FUNCTION_BLOCK DataConversionDecorator IMPLEMENTS ITF_Analogue
VAR
	wrappee : ITF_Analogue;
END_VAR

METHOD GetValue : INT
IF (THIS^.wrappee <> 0) THEN
  GetValue := THIS^.wrappee.GetValue() + 0.9;
END_IF
END_METHOD

END_FUNCTION_BLOCK

(* stored: Version 1.1.0.1, ProductVersion 3.1.4024.12
   POU DataConversionDecorator: Id {4b1d2179-15d5-4bf4-bc8e-05c702dbfa59}, SpecialFunc None
   Method GetValue: Id {643484a3-ba6c-4b4b-9e12-d59a094794f0} *)
